DATA_BLOCK "Db16070_ControlloSpessore"
{ DB_Accessible_From_OPC_UA := 'FALSE' ;
 S7_Optimized_Access := 'FALSE' }
VERSION : 0.2
"Fb936_ControlloSpessore_v11"

BEGIN
   I_ParametriCntrolloSpessore.PosizioneCentroVentosa := 1930.0;
   I_ParametriCntrolloSpessore.RangeControllo := 80.0;
   I_ParametriCntrolloSpessore.RangeRallenta := 500.0;
   I_ParametriCntrolloSpessore.nLettureConsecutiveAllarme := 15.0;
   I_ParametriCntrolloSpessore.SpessoreMassimo := 1.0;
   I_ParametriCntrolloSpessore.OvrTrasfertPerpassaggio := 100.0;
   I_ParametriCntrolloSpessore.DisabilitaControllo := FALSE;
   I_ParametriCntrolloSpessore.SpessoreDiscoRiferimento := 2.98;
   I_ParametriCntrolloSpessore.AbilitaTaratura := FALSE;
   Pinza.OvrAutoOld := 0.0;
   Pinza.OvrManOld := 0.0;
   aBaseline[0] := 0.0;
   aBaseline[1] := 0.0;
   aBaseline[2] := 0.0;
   aBaseline[3] := 0.0;
   aBaseline[4] := 0.0;
   aBaseline[5] := 0.0;
   aBaseline[6] := 0.0;
   aBaseline[7] := 0.0;
   aBaseline[8] := 0.0;
   aBaseline[9] := 0.0;
   aBaseline[10] := 0.0;
   aBaseline[11] := 0.0;
   aBaseline[12] := 0.0;
   aBaseline[13] := 0.0;
   aBaseline[14] := 0.0;
   aBaseline[15] := 0.0;
   aBaseline[16] := 0.0;
   aBaseline[17] := 0.0;
   aBaseline[18] := 0.0;
   aBaseline[19] := 0.0;
   aBaseline[20] := 0.0;
   aBaseline[21] := 0.0;
   aBaseline[22] := 0.0;
   aBaseline[23] := 0.0;
   aBaseline[24] := 0.0;
   aBaseline[25] := 0.0;
   aBaseline[26] := 0.0;
   aBaseline[27] := 0.0;
   aBaseline[28] := 0.0;
   aBaseline[29] := 0.0;
   aBaseline[30] := 0.0;
   aBaseline[31] := 0.0;
   aBaseline[32] := 0.0;
   aBaseline[33] := 0.0;
   aBaseline[34] := 0.0;
   aBaseline[35] := 0.0;
   aBaseline[36] := 0.0;
   aBaseline[37] := 0.0;
   aBaseline[38] := 0.0;
   aBaseline[39] := 0.0;
   aBaseline[40] := 0.0;
   aBaseline[41] := 0.0;
   aBaseline[42] := 0.0;
   aBaseline[43] := 0.0;
   aBaseline[44] := 0.0;
   aBaseline[45] := 0.0;
   aBaseline[46] := 0.0;
   aBaseline[47] := 0.0;
   aBaseline[48] := 0.0;
   aBaseline[49] := 0.0;
   aBaseline[50] := 0.0;
   aBaseline[51] := 0.0;
   aBaseline[52] := 0.0;
   aBaseline[53] := 0.0;
   aBaseline[54] := 0.0;
   aBaseline[55] := 0.0;
   aBaseline[56] := 0.0;
   aBaseline[57] := 0.0;
   aBaseline[58] := 0.0;
   aBaseline[59] := 0.0;
   aBaseline[60] := 0.0;
   aBaseline[61] := 0.0;
   aBaseline[62] := 0.0;
   aBaseline[63] := 0.0;
   aBaseline[64] := 0.0;
   aBaseline[65] := 0.0;
   aBaseline[66] := 0.0;
   aBaseline[67] := 0.0;
   aBaseline[68] := 0.0;
   aBaseline[69] := 0.0;
   aBaseline[70] := 0.0;
   aBaseline[71] := 0.0;
   aBaseline[72] := 0.0;
   aBaseline[73] := 0.0;
   aBaseline[74] := 0.0;
   aBaseline[75] := 0.0;
   aBaseline[76] := 0.0;
   aBaseline[77] := 0.0;
   aBaseline[78] := 0.0;
   aBaseline[79] := 0.0;
   aBaseline[80] := 0.0;
   aBaseline[81] := 0.0;
   aBaseline[82] := 0.0;
   aBaseline[83] := 0.0;
   aBaseline[84] := 0.0;
   aBaseline[85] := 0.0;
   aBaseline[86] := 0.0;
   aBaseline[87] := 0.0;
   aBaseline[88] := 0.0;
   aBaseline[89] := 0.0;
   aBaseline[90] := 0.0;
   aBaseline[91] := 0.0;
   aBaseline[92] := 0.0;
   aBaseline[93] := 0.0;
   aBaseline[94] := 0.0;
   aBaseline[95] := 0.0;
   aBaseline[96] := 0.0;
   aBaseline[97] := 0.0;
   aBaseline[98] := 0.0;
   aBaseline[99] := 0.0;
   aBaseline[100] := 0.0;
   aBaseline[101] := 0.0;
   aBaseline[102] := 0.0;
   aBaseline[103] := 0.0;
   aBaseline[104] := 0.0;
   aBaseline[105] := 0.0;
   aBaseline[106] := 0.0;
   aBaseline[107] := 0.0;
   aBaseline[108] := 0.0;
   aBaseline[109] := 0.0;
   aBaseline[110] := 0.0;
   aBaseline[111] := 0.0;
   aBaseline[112] := 0.0;
   aBaseline[113] := 0.0;
   aBaseline[114] := 0.0;
   aBaseline[115] := 0.0;
   aBaseline[116] := 0.0;
   aBaseline[117] := 0.0;
   aBaseline[118] := 0.0;
   aBaseline[119] := 0.0;
   aBaseline[120] := 0.0;
   aBaseline[121] := 0.0;
   aBaseline[122] := 0.0;
   aBaseline[123] := 0.0;
   aBaseline[124] := 0.0;
   aBaseline[125] := 0.0;
   aBaseline[126] := 0.0;
   aBaseline[127] := 0.0;
   aBaseline[128] := 0.0;
   aBaseline[129] := 0.0;
   aBaseline[130] := 0.0;
   aBaseline[131] := 0.0;
   aBaseline[132] := 0.0;
   aBaseline[133] := 0.0;
   aBaseline[134] := 0.0;
   aBaseline[135] := 0.0;
   aBaseline[136] := 0.0;
   aBaseline[137] := 0.0;
   aBaseline[138] := 0.0;
   aBaseline[139] := 0.0;
   aBaseline[140] := 0.0;
   aBaseline[141] := 0.0;
   aBaseline[142] := 0.0;
   aBaseline[143] := 0.0;
   aBaseline[144] := 0.0;
   aBaseline[145] := 0.0;
   aBaseline[146] := 0.0;
   aBaseline[147] := 0.0;
   aBaseline[148] := 0.0;
   aBaseline[149] := 0.0;
   aBaseline[150] := 0.0;
   aBaseline[151] := 0.0;
   aBaseline[152] := 0.0;
   aBaseline[153] := 0.0;
   aBaseline[154] := 0.0;
   aBaseline[155] := 0.0;
   aBaseline[156] := 0.0;
   aBaseline[157] := 0.0;
   aBaseline[158] := 0.0;
   aBaseline[159] := 0.0;
   aBaseline[160] := 0.0;
   aBaseline[161] := 0.0;
   aBaseline[162] := 0.0;
   aBaseline[163] := 0.0;
   aBaseline[164] := 0.0;
   aBaseline[165] := 0.0;
   aBaseline[166] := 0.0;
   aBaseline[167] := 0.0;
   aBaseline[168] := 0.0;
   aBaseline[169] := 0.0;
   aBaseline[170] := 0.0;
   aBaseline[171] := 0.0;
   aBaseline[172] := 0.0;
   aBaseline[173] := 0.0;
   aBaseline[174] := 0.0;
   aBaseline[175] := 0.0;
   aBaseline[176] := 0.0;
   aBaseline[177] := 0.0;
   aBaseline[178] := 0.0;
   aBaseline[179] := 0.0;
   aBaseline[180] := 0.0;
   aBaseline[181] := 0.0;
   aBaseline[182] := 0.0;
   aBaseline[183] := 0.0;
   aBaseline[184] := 0.0;
   aBaseline[185] := 0.0;
   aBaseline[186] := 0.0;
   aBaseline[187] := 0.0;
   aBaseline[188] := 0.0;
   aBaseline[189] := 0.0;
   aBaseline[190] := 0.0;
   aBaseline[191] := 0.0;
   aBaseline[192] := 0.0;
   aBaseline[193] := 0.0;
   aBaseline[194] := 0.0;
   aBaseline[195] := 0.0;
   aBaseline[196] := 0.0;
   aBaseline[197] := 0.0;
   aBaseline[198] := 0.0;
   aBaseline[199] := 0.0;
   aBaseline[200] := 0.0;
   OldDirLavoro := 2;
   AuxFpCambioDirezione := FALSE;

END_DATA_BLOCK

